NETWORK
TITLE = ---- Final
////////////////////////////////////////////////////////////////////////////////////////
////////////////////////////////////////////////////////////////////////////////////////
////////////////////////////////////////////////////////////////////////////////////////
// Se acabo el evento
Final_EventoRecibido_RefrescoUT:NOP   0;
      L     #P_Eventos;  // Recupero por donde voy en la lista de eventos
      LAR2;  // Regreso a buscar el siguiente evento
      JU    FinBucle_EventosRecibidos;



NETWORK
TITLE = Guardar Datos - Evento MOVE - Mover UT de Mesa // 08 02 2017
GuardarDatos_EventoRecibido_MOVE:NOP   0;

/////////////////////////////////////////////////////////////////////////
/////////////////////////////////////////////////////////////////////////
/////////////////////////////////////////////////////////////////////////
// --- Guardar Datos del Evento Recibido


/////////////////////////////////////////////////////////////////////////
/////////////////////////////////////////////////////////////////////////
/////////////////////////////////////////////////////////////////////////
// --- Control de Mesa Recibida
      L     #AtributosDeUTs.MesaActual;  // Ver que mesa es
      L     "CTE_OffsetMesa";
      -I;
      T     #VarTempUTs.MesaActual;

      L     #VarTempUTs.MesaActual;  // Comprobar el numero de mesa
      L     1;  // No menor de 1
      <I;  // No es correcto
      JC    Final_EventoRecibido_MOVE;
      L     #VarTempUTs.MesaActual;
      L     "CTE_MaxMesas";  // No mayor que el parametro
      >I;  // No es correcto
      JC    Final_EventoRecibido_MOVE;


///////////////////////////////////////////////////////////////////////////////
// --- Control de McKey Recibido
      L     #AtributosDeUTs.Mckey;  // Se ha recibido Mckey = 0
      L     0;  // No se puede Crear
      ==D;
      JC    Final_EventoRecibido_MOVE;


///////////////////////////////////////////////////////////////////////////////
// --- Busca el Mckey Recibido, comprobar que existe

      CALL  "FC720_BuscarUT_EnMesa"
      ( Mckey      := #AtributosDeUTs.Mckey,
        MesaActual := #VarTempUTs.MesaActual,
        NumeroUT   := #VarTempUTs.NumeroUT
      );

      L     #VarTempUTs.NumeroUT;
      L     0;
      ==I;  // No Existe UT ?
      JC    Final_EventoRecibido_MOVE;



NETWORK
TITLE = ---- Accion del Evento
///////////////////////////////////////////////////////////////////////////////
///////////////////////////////////////////////////////////////////////////////
///////////////////////////////////////////////////////////////////////////////
// --- Guardar Respuesta

      SET;
      L     "DB812_UTs_Control".UT[#VarTempUTs.NumeroUT].MesaActual;
      L     #AtributosDeUTs.MesaActual;
      <>I;  // Esta en Mesa diferente ?
      JC    Final_EventoRecibido_MOVE;

      SET;  // Realizada la peticion de Cambio de Mesa ?
      AN    "DB812_UTs_Control".UT[#VarTempUTs.NumeroUT].EventosDeCambioDeMesa.PeticionCambiarUTDeMesa;
      JC    Final_EventoRecibido_MOVE;


///////////////////////////////////////////////////////////////////////////////
///////////////////////////////////////////////////////////////////////////////
///////////////////////////////////////////////////////////////////////////////
// --- Orden Recibida guardarla en la UT

      SET;  // OK Cambiar UT de Mesa Final
      A     #AtributosDeUTs.CambiarUTDeMesa.OK;
      A     #AtributosDeUTs.CambiarUTDeMesa.Final;
      S     "DB812_UTs_Control".UT[#VarTempUTs.NumeroUT].EventosDeCambioDeMesa.OKCambiarUTDeMesaFinal;

      SET;  // OK Cambiar UT de Mesa Inicio
      A     #AtributosDeUTs.CambiarUTDeMesa.OK;
      A     #AtributosDeUTs.CambiarUTDeMesa.Inicio;
      S     "DB812_UTs_Control".UT[#VarTempUTs.NumeroUT].EventosDeCambioDeMesa.OKCambiarUTDeMesaInicio;

      SET;  // NOK Cambiar UT de Mesa
      A     #AtributosDeUTs.CambiarUTDeMesa.NOK;
      S     "DB812_UTs_Control".UT[#VarTempUTs.NumeroUT].EventosDeCambioDeMesa.NOKCambiarUTDeMesa;


///////////////////////////////////////////////////////////////////////////////
      JU    Final_EventoRecibido_MOVE;



NETWORK
TITLE = ---- Final
///////////////////////////////////////////////////////////////////////////////
///////////////////////////////////////////////////////////////////////////////
///////////////////////////////////////////////////////////////////////////////
// Se acabo el evento
Final_EventoRecibido_MOVE:NOP   0;
      L     #P_Eventos;  // Recupero por donde voy en la lista de eventos
      LAR2;
      JU    FinBucle_EventosRecibidos;



NETWORK
TITLE = Guardar Datos - Evento DEMB - Datos de EmBandejado de la UT // Fecha 07 06 2017
GuardarDatos_EventoRecibido_DEMB:NOP   0;

/////////////////////////////////////////////////////////////////////////
/////////////////////////////////////////////////////////////////////////
/////////////////////////////////////////////////////////////////////////
// --- Guardar Datos del Evento Recibido


/////////////////////////////////////////////////////////////////////////
/////////////////////////////////////////////////////////////////////////
/////////////////////////////////////////////////////////////////////////
// --- Control de Mesa Recibida
      L     #AtributosDeUTs.MesaActual;
      L     0;
      ==I;
      JC    FinControlMesa_EventoRecibido_DEMB;

      L     #AtributosDeUTs.MesaActual;  // Ver que mesa es
      L     "CTE_OffsetMesa";
      -I;
      T     #VarTempUTs.MesaActual;

      L     #VarTempUTs.MesaActual;  // Comprobar el numero de mesa
      L     1;  // No menor de 1
      <I;  // No es correcto
      JC    Final_EventoRecibido_DEMB;
      L     #VarTempUTs.MesaActual;
      L     "CTE_MaxMesas";  // No mayor que el parametro
      >I;  // No es correcto
      JC    Final_EventoRecibido_DEMB;

/////////////////////////////////////////////////////////////////////////
FinControlMesa_EventoRecibido_DEMB:NOP   0;


/////////////////////////////////////////////////////////////////////////
/////////////////////////////////////////////////////////////////////////
/////////////////////////////////////////////////////////////////////////
// --- Control de Mckey Recibido
      L     #AtributosDeUTs.Mckey;  // Se ha recibido Mckey = 0
      L     0;  // No se puede Crear
      ==D;
      JC    Final_EventoRecibido_DEMB;


/////////////////////////////////////////////////////////////////////////
/////////////////////////////////////////////////////////////////////////
/////////////////////////////////////////////////////////////////////////
// --- Comprobar que Existe una UT
      CALL  "FC720_BuscarUT_EnMesa"
      ( Mckey      := #AtributosDeUTs.Mckey,
        MesaActual := #VarTempUTs.MesaActual,
        NumeroUT   := #VarTempUTs.NumeroUT
      );

      L     #VarTempUTs.NumeroUT;
      L     0;
      ==I;  // No Existe UT ?
      JC    Final_EventoRecibido_DEMB;



NETWORK
TITLE = ---- Accion del Evento
/////////////////////////////////////////////////////////////////////////
/////////////////////////////////////////////////////////////////////////
/////////////////////////////////////////////////////////////////////////
// Guardar Respuesta


      L     #AtributosDeUTs.QUBIQA_NumeroBulto;  // Numero de Bulto
      T     "DB820_UTs_DatosQUBIQA".UT[#VarTempUTs.NumeroUT].NumeroDeBulto;
      L     #AtributosDeUTs.QUBIQA_TotalBultos;  // Numero de Bultos
      T     "DB820_UTs_DatosQUBIQA".UT[#VarTempUTs.NumeroUT].TotalBultos;

      CALL  BLKMOV
      ( SRCBLK  := #AtributosDeUTs.QUBIQA_PID,
        RET_VAL := #ReturnValor,
        DSTBLK  := "DB820_UTs_DatosQUBIQA".UT[#VarTempUTs.NumeroUT].PID
      );  // Guardar el PID

      JU    Final_EventoRecibido_DEMB;



NETWORK
TITLE = ---- Final
/////////////////////////////////////////////////////////////////////////
/////////////////////////////////////////////////////////////////////////
/////////////////////////////////////////////////////////////////////////
// Se acabo el evento
Final_EventoRecibido_DEMB:NOP   0;
      L     #P_Eventos;  // Recupero por donde voy en la lista de eventos
      LAR2;
      JU    FinBucle_EventosRecibidos;



NETWORK
TITLE = ////////////////////////////////////////////////////////////////////////////////////////////////////////////

NETWORK
TITLE = Evento CSTA - Notificacion de cambio de Estado de un dispositivo
// Analisis del evento
// - Inicializa variables de los atributos del Evento
// - Buscar Atributos o Final del Evento
// - Guardar datos del Evento
//   - Si es tipo CCPIF (50)
//   - Si es tipo CBOX (40)
//   - Si es tipo Mesa (60)
//   - Si es tipo Maquina (70)
// Analisis de los atributos de los eventos
// - Mirar que atributo del Evento es ?
// - Distribuir a recoger los datos del Evento
// - Recoger el Atributo Tipo de Dispositivo
// - Recoger el Atributo Numero de Dispositivo
// - Recoger el Atributo Nuevo Estado del Dispositivo
GuardarDatos_EventoRecibido_CSTA:NOP   0;

/////////////////////////////////////////////////////////////////////////
/////////////////////////////////////////////////////////////////////////
/////////////////////////////////////////////////////////////////////////
// --- Guardar Datos del Evento Recibido


/////////////////////////////////////////////////////////////////////////
/////////////////////////////////////////////////////////////////////////
/////////////////////////////////////////////////////////////////////////
// --- Repartir segun tipo de dispositivo: CCPIF, CBOX, Mesa ....

      SET;  // Es CCPIF
      L     #AtributosDeDispositivos.Tipo;
      L     50;
      ==I;
      JC    DispositivosCCPIF_EventoRecibido_CSTA;

      SET;  // Es CBOX
      L     #AtributosDeDispositivos.Tipo;
      L     40;
      ==I;
      JC    DispositivosCBOX_EventoRecibido_CSTA;

      SET;  // Es Mesa
      L     #AtributosDeDispositivos.Tipo;
      L     60;
      ==I;
      JC    DispositivosMesa_EventoRecibido_CSTA;

      SET;  // Es Baliza
      L     #AtributosDeDispositivos.Tipo;
      L     1000;
      ==I;
      JC    DispositivosBaliza_EventoRecibido_CSTA;

/////////////////////////////////////////////////////////////////////////
/////////////////////////////////////////////////////////////////////////
/////////////////////////////////////////////////////////////////////////

      SET;  // Es Llave
      L     #AtributosDeDispositivos.Tipo;
      L     1001;
      ==I;
      JC    DispositivosLlave_EventoRecibido_CSTA;

      SET;  // Es Seta
      L     #AtributosDeDispositivos.Tipo;
      L     1002;
      ==I;
      JC    DispositivosSeta_EventoRecibido_CSTA;

      SET;  // Es Barrera
      L     #AtributosDeDispositivos.Tipo;
      L     1003;
      ==I;
      JC    DispositivosBarrera_EventoRecibido_CSTA;

      SET;  // Es Puerta
      L     #AtributosDeDispositivos.Tipo;
      L     1004;
      ==I;
      JC    DispositivosPuerta_EventoRecibido_CSTA;

      SET;  // Es Linea de Potencia
      L     #AtributosDeDispositivos.Tipo;
      L     1005;
      ==I;
      JC    DispositivosLineaPotencia_EventoRecibido_CSTA;


/////////////////////////////////////////////////////////////////////////
/////////////////////////////////////////////////////////////////////////
/////////////////////////////////////////////////////////////////////////
// Es Maquina De 70 ... 99
      SET;
      A(;
      L     #AtributosDeDispositivos.Tipo;
      L     70;
      >=I;
      );
      A(;
      SET;
      L     #AtributosDeDispositivos.Tipo;
      L     99;
      <=I;
      );
      JC    DispositivosMaquina_EventoRecibido_CSTA;


/////////////////////////////////////////////////////////////////////////
/////////////////////////////////////////////////////////////////////////
/////////////////////////////////////////////////////////////////////////
// --- No es ningun Tipo de Dispositivo Esperado
      JU    Final_EventoRecibido_CSTA;



NETWORK
TITLE = ---- Accion del Evento --> Notificacion de cambio de Estado de CCPIF
///////////////////////////////////////////////////////////////////////////////
///////////////////////////////////////////////////////////////////////////////
///////////////////////////////////////////////////////////////////////////////
// --- Tipo CCPIF
DispositivosCCPIF_EventoRecibido_CSTA:NOP   0;


///////////////////////////////////////////////////////////////////////////////
// --- Comprobacion del Numero de Dispositivo
      L     #AtributosDeDispositivos.Numero;  // Comprobacion del numero de CCPIF
      L     "CTE_OffsetCCPIF";
      -I;
      L     1;
      <>I;  // Numero de CCPIF incorrecto
      JC    Final_EventoRecibido_CSTA;


///////////////////////////////////////////////////////////////////////////////
// --- Guardar el Cambio de Estado Recibido
      L     #AtributosDeDispositivos.NuevoEstado;  // EstadoDispo + 260 = Recibido Evento de Cambio de Estado
      L     260;  // Orden a guardar en el DB
      +I;
      T     "DB830_Dispositivos".Dispositivos[0].EstadoRecepcionEvento;


///////////////////////////////////////////////////////////////////////////////
// --- Finalizar
      JU    Final_EventoRecibido_CSTA;



NETWORK
TITLE = ---- Accion del Evento --> Notificacion de cambio de Estado de CBOX
///////////////////////////////////////////////////////////////////////////////
///////////////////////////////////////////////////////////////////////////////
///////////////////////////////////////////////////////////////////////////////
// --- Tipo CBOX
DispositivosCBOX_EventoRecibido_CSTA:NOP   0;


///////////////////////////////////////////////////////////////////////////////
// --- Comprobacion del Numero de Dispositivo
      L     #AtributosDeDispositivos.Numero;  // Comprobacion del numero de CCPIF
      L     100;
      /I;
      L     "CTE_OffsetCCPIF";
      -I;
      L     1;
      <>I;  // Numero de CCPIF incorrecto
      JC    Final_EventoRecibido_CSTA;


      L     #AtributosDeDispositivos.Numero;  // Calculo del numero de CBOX
      L     100;
      MOD;  // Var verlo en la DB_Dispositivos
      T     #VarTempDispositivos.Numero;

      L     #VarTempDispositivos.Numero;  // Comprobacion del numero de CBOX
      L     1;  // Es menor de 1
      <I;  // No es correcto el numero de CBOX
      JC    Final_EventoRecibido_CSTA;
      L     #VarTempDispositivos.Numero;
      L     "CTE_MaxDispositivos";  // Si es mayor que el parametro
      >I;  // No es correcto el numero de CBOX
      JC    Final_EventoRecibido_CSTA;


///////////////////////////////////////////////////////////////////////////////
// --- Guardar el Cambio de Estado Recibido
      L     #AtributosDeDispositivos.NuevoEstado;  // EstadoDispo + 260 = Recibido Evento de Cambio de Estado
      L     260;  // Orden a guardar en el DB
      +I;
      T     "DB830_Dispositivos".Dispositivos[#VarTempDispositivos.Numero].EstadoRecepcionEvento;


///////////////////////////////////////////////////////////////////////////////
// --- Finalizar
      JU    Final_EventoRecibido_CSTA;



NETWORK
TITLE = ---- Accion del Evento --> Notificacion de cambio de Estado de Mesa
///////////////////////////////////////////////////////////////////////////////
///////////////////////////////////////////////////////////////////////////////
///////////////////////////////////////////////////////////////////////////////
// --- Tipo Mesa
DispositivosMesa_EventoRecibido_CSTA:NOP   0;


///////////////////////////////////////////////////////////////////////////////
// --- Comprobacion del Numero de Dispositivo
      L     #AtributosDeDispositivos.Numero;  // Ver que mesa es
      L     "CTE_OffsetMesa";
      -I;
      T     #VarTempDispositivos.Numero;

      L     #VarTempDispositivos.Numero;  // Comprobar el numero de mesa
      L     1;  // No menor de 1
      <I;  // No es correcto
      JC    Final_EventoRecibido_CSTA;
      L     #VarTempDispositivos.Numero;
      L     "CTE_MaxMesas";  // No meyor que el parametro
      >I;  // No es correcto
      JC    Final_EventoRecibido_CSTA;


///////////////////////////////////////////////////////////////////////////////
// --- Guardar el Cambio de Estado Recibido
      L     #AtributosDeDispositivos.NuevoEstado;  // EstadoDispo + 260 = Recibido Evento de Cambio de Estado
      L     260;  // Orden a guardar en el DB
      +I;
      T     "DB831_Mesas".Mesas[#VarTempDispositivos.Numero].EstadoRecepcionEvento;


///////////////////////////////////////////////////////////////////////////////
// --- Habilitado o DesHabilitado el Dispositivo
      SET;
      L     #AtributosDeDispositivos.Habilitado;
      L     2001;  // Habitar Disposito = 0
      ==I;
      R     "DB831_Mesas".Mesas[#VarTempDispositivos.Numero].Memorias.DesHabilitado;

      SET;
      L     #AtributosDeDispositivos.Habilitado;
      L     2002;  // DesHabitar Disposito = 1
      ==I;
      S     "DB831_Mesas".Mesas[#VarTempDispositivos.Numero].Memorias.DesHabilitado;


///////////////////////////////////////////////////////////////////////////////
// Prioridad  - 1...x
      SET;
      L     #AtributosDeDispositivos.Prioridad;
      L     0;
      ==I;
      JC    SinPrioridadMesa_EventoRecibido_CSTA;

      L     #AtributosDeDispositivos.Prioridad;
      T     "DB831_Mesas".Mesas[#VarTempDispositivos.Numero].Prioridad;

SinPrioridadMesa_EventoRecibido_CSTA:NOP   0;


///////////////////////////////////////////////////////////////////////////////
// --- Fecha: 08 02 2017
// --- Motivo para la pantalla del Error envio por el JDT
      SET;
      L     #LonguitudTextoRecibido;
      L     0;
      ==I;  // Existe Motivo de Error en Mesa Enviado por el JDT
      JC    SinMotivoDeErrorDelJdT_EventoRecibido_CSTA;

      CALL  BLKMOV
      ( SRCBLK  := #AtributosDeDispositivos.MotivoDelError,
        RET_VAL := #ReturnValor,
        DSTBLK  := "DB907_TextoErrorJdT".Mesa[#VarTempDispositivos.Numero]
      );

SinMotivoDeErrorDelJdT_EventoRecibido_CSTA:NOP   0;


///////////////////////////////////////////////////////////////////////////////
// --- Finalizar
      JU    Final_EventoRecibido_CSTA;



NETWORK
TITLE = ---- Accion del Evento --> Notificacion de cambio de Estado de Maquina
///////////////////////////////////////////////////////////////////////////////
///////////////////////////////////////////////////////////////////////////////
///////////////////////////////////////////////////////////////////////////////
// --- Tipo Maquina
DispositivosMaquina_EventoRecibido_CSTA:NOP   0;


///////////////////////////////////////////////////////////////////////////////
// --- Comprobacion del Numero de Dispositivo
      L     #AtributosDeDispositivos.Numero;  // Ver que mesa es
      L     "CTE_OffsetMesa";
      -I;
      T     #VarTempDispositivos.Numero;

      L     #VarTempDispositivos.Numero;  // Comprobar el numero de maquina
      L     1;  // No menor de 1
      <I;  // No es correcto
      JC    Final_EventoRecibido_CSTA;
      L     #VarTempDispositivos.Numero;
      L     "CTE_MaxMesas";  // No meyor que el parametro
      >I;  // No es correcto
      JC    Final_EventoRecibido_CSTA;


///////////////////////////////////////////////////////////////////////////////
// --- Guardar el Cambio de Estado Recibido

      L     #AtributosDeDispositivos.NuevoEstado;  // EstadoDispo + 260 = Recibido Evento de Cambio de Estado
      L     260;  // Orden a guardar en el DB
      +I;
      T     "DB832_Maquinas".Maquinas[#VarTempDispositivos.Numero].EstadoRecepcionEvento;


///////////////////////////////////////////////////////////////////////////////
// --- Habilitado o DesHabilitado
      SET;
      L     #AtributosDeDispositivos.Habilitado;
      L     2001;  // Habitar Disposito = 0
      ==I;
      R     "DB832_Maquinas".Maquinas[#VarTempDispositivos.Numero].Memorias.DesHabilitado;

      SET;
      L     #AtributosDeDispositivos.Habilitado;
      L     2002;  // DesHabitar Disposito = 1
      ==I;
      S     "DB832_Maquinas".Maquinas[#VarTempDispositivos.Numero].Memorias.DesHabilitado;


///////////////////////////////////////////////////////////////////////////////
// Prioridad  - 1...x
      SET;
      L     #AtributosDeDispositivos.Prioridad;
      L     0;
      ==I;
      JC    SinPrioridadMaquina_EventoRecibido_CSTA;

      L     #AtributosDeDispositivos.Prioridad;
      T     "DB832_Maquinas".Maquinas[#VarTempDispositivos.Numero].Prioridad;

SinPrioridadMaquina_EventoRecibido_CSTA:NOP   0;


///////////////////////////////////////////////////////////////////////////////
// Finalizar
      JU    Final_EventoRecibido_CSTA;



NETWORK
TITLE = ---- Accion del Evento --> Notificacion de cambio de Estado de Baliza
///////////////////////////////////////////////////////////////////////////////
///////////////////////////////////////////////////////////////////////////////
///////////////////////////////////////////////////////////////////////////////
// --- Tipo Baliza
DispositivosBaliza_EventoRecibido_CSTA:NOP   0;


///////////////////////////////////////////////////////////////////////////////
// --- Comprobacion del Numero de Dispositivo
      L     #AtributosDeDispositivos.Numero;  // Ver que Baliza es
      L     "CTE_OffsetMesa";
      -I;
      T     #VarTempDispositivos.Numero;

      L     #VarTempDispositivos.Numero;  // Comprobar el numero de Baliza
      L     1;  // No menor de 1
      <I;  // No es correcto
      JC    Final_EventoRecibido_CSTA;
      L     #VarTempDispositivos.Numero;
      L     "CTE_MaxDispositivosBaliza";  // No meyor que el parametro
      >I;  // No es correcto
      JC    Final_EventoRecibido_CSTA;


///////////////////////////////////////////////////////////////////////////////
// --- Guardar el Cambio de Estado Recibido

      CALL  BLKMOV
      ( SRCBLK  := "DB839_DispositivosVarios".DispoBaliza[#VarTempDispositivos.Numero],
        RET_VAL := #ReturnValor,
        DSTBLK  := #VarTempDispositivos.Baliza
      );

      SET;  // Reseteo para actualizar
      R     #VarTempDispositivos.Baliza.Sonoro;
      R     #VarTempDispositivos.Baliza.Verde;
      R     #VarTempDispositivos.Baliza.Rojo;
      R     #VarTempDispositivos.Baliza.Amarillo;
      R     #VarTempDispositivos.Baliza.Azul;


      SET;  // Sonoro
      A     #AtributosDeDispositivos.BalizaColor.Sonoro;
      S     #VarTempDispositivos.Baliza.Sonoro;

      SET;  // Verde
      A     #AtributosDeDispositivos.BalizaColor.Verde;
      S     #VarTempDispositivos.Baliza.Verde;

      SET;  // Rojo
      A     #AtributosDeDispositivos.BalizaColor.Rojo;
      S     #VarTempDispositivos.Baliza.Rojo;

      SET;  // Amarillo
      A     #AtributosDeDispositivos.BalizaColor.Amarillo;
      S     #VarTempDispositivos.Baliza.Amarillo;

      SET;  // Azul
      A     #AtributosDeDispositivos.BalizaColor.Azul;
      S     #VarTempDispositivos.Baliza.Azul;

      SET;  // Peticion de Estado
      S     #VarTempDispositivos.Baliza.RefrescoDatos;

      CALL  BLKMOV
      ( SRCBLK  := #VarTempDispositivos.Baliza,
        RET_VAL := #ReturnValor,
        DSTBLK  := "DB839_DispositivosVarios".DispoBaliza[#VarTempDispositivos.Numero]
      );


///////////////////////////////////////////////////////////////////////////////
// Finalizar
      JU    Final_EventoRecibido_CSTA;



NETWORK
TITLE = ---- Accion del Evento --> Notificacion de cambio de Estado de Llave
///////////////////////////////////////////////////////////////////////////////
///////////////////////////////////////////////////////////////////////////////
///////////////////////////////////////////////////////////////////////////////
// --- Tipo Llave
DispositivosLlave_EventoRecibido_CSTA:NOP   0;


///////////////////////////////////////////////////////////////////////////////
// --- Comprobacion del Numero de Dispositivo
      L     #AtributosDeDispositivos.Numero;  // Ver que Llave es
      L     "CTE_OffsetMesa";
      -I;
      T     #VarTempDispositivos.Numero;

      L     #VarTempDispositivos.Numero;  // Comprobar el numero de Llave
      L     1;  // No menor de 1
      <I;  // No es correcto
      JC    Final_EventoRecibido_CSTA;
      L     #VarTempDispositivos.Numero;
      L     "CTE_MaxDispositivosLlave";  // No meyor que el parametro
      >I;  // No es correcto
      JC    Final_EventoRecibido_CSTA;


///////////////////////////////////////////////////////////////////////////////
// --- Guardar el Cambio de Estado Recibido

      SET;
      S     "DB839_DispositivosVarios".DispoLlave[#VarTempDispositivos.Numero].Habilitado;  // Por defecto DesHabilitado

      L     #AtributosDeDispositivos.Habilitado;
      L     2001;  // Nuevo estado - Habilitado SI ?
      ==I;
      JC    HabilitadaLlave_EventoRecibido_CSTA;

      SET;
      R     "DB839_DispositivosVarios".DispoLlave[#VarTempDispositivos.Numero].Habilitado;

HabilitadaLlave_EventoRecibido_CSTA:NOP   0;

      SET;
      S     "DB839_DispositivosVarios".DispoLlave[#VarTempDispositivos.Numero].RefrescoDatos;  // Peticion de Refresco de datos


///////////////////////////////////////////////////////////////////////////////
// Finalizar
      JU    Final_EventoRecibido_CSTA;



NETWORK
TITLE = ---- Accion del Evento --> Notificacion de cambio de Estado de Seta
///////////////////////////////////////////////////////////////////////////////
///////////////////////////////////////////////////////////////////////////////
///////////////////////////////////////////////////////////////////////////////
// --- Tipo Seta
DispositivosSeta_EventoRecibido_CSTA:NOP   0;


///////////////////////////////////////////////////////////////////////////////
// --- Comprobacion del Numero de Dispositivo
      L     #AtributosDeDispositivos.Numero;  // Ver que Seta es
      L     "CTE_OffsetMesa";
      -I;
      T     #VarTempDispositivos.Numero;

      L     #VarTempDispositivos.Numero;  // Comprobar el numero de Seta
      L     1;  // No menor de 1
      <I;  // No es correcto
      JC    Final_EventoRecibido_CSTA;
      L     #VarTempDispositivos.Numero;
      L     "CTE_MaxDispositivosSeta";  // No meyor que el parametro
      >I;  // No es correcto
      JC    Final_EventoRecibido_CSTA;


///////////////////////////////////////////////////////////////////////////////
// --- Guardar el Cambio de Estado Recibido

      SET;
      S     "DB839_DispositivosVarios".DispoSeta[#VarTempDispositivos.Numero].Habilitado;  // Por defecto DesHabilitado

      L     #AtributosDeDispositivos.Habilitado;
      L     2001;  // Nuevo estado - Habilitado SI ?
      ==I;
      JC    HabilitadaSeta_EventoRecibido_CSTA;

      SET;
      R     "DB839_DispositivosVarios".DispoSeta[#VarTempDispositivos.Numero].Habilitado;

HabilitadaSeta_EventoRecibido_CSTA:NOP   0;

      SET;
      S     "DB839_DispositivosVarios".DispoSeta[#VarTempDispositivos.Numero].RefrescoDatos;  // Peticion de Refresco de datos


///////////////////////////////////////////////////////////////////////////////
// Finalizar
      JU    Final_EventoRecibido_CSTA;



NETWORK
TITLE = ---- Accion del Evento --> Notificacion de cambio de Estado de Barrera
///////////////////////////////////////////////////////////////////////////////
///////////////////////////////////////////////////////////////////////////////
///////////////////////////////////////////////////////////////////////////////
// --- Tipo Barrera
DispositivosBarrera_EventoRecibido_CSTA:NOP   0;


///////////////////////////////////////////////////////////////////////////////
// --- Comprobacion del Numero de Dispositivo
      L     #AtributosDeDispositivos.Numero;  // Ver que Barrera es
      L     "CTE_OffsetMesa";
      -I;
      T     #VarTempDispositivos.Numero;

      L     #VarTempDispositivos.Numero;  // Comprobar el numero de Barrera
      L     1;  // No menor de 1
      <I;  // No es correcto
      JC    Final_EventoRecibido_CSTA;
      L     #VarTempDispositivos.Numero;
      L     "CTE_MaxDispositivosBarrera";  // No meyor que el parametro
      >I;  // No es correcto
      JC    Final_EventoRecibido_CSTA;


///////////////////////////////////////////////////////////////////////////////
// --- Guardar el Cambio de Estado Recibido

      SET;
      S     "DB839_DispositivosVarios".DispoBarrera[#VarTempDispositivos.Numero].Habilitado;  // Por defecto DesHabilitado

      L     #AtributosDeDispositivos.Habilitado;
      L     2001;  // Nuevo estado - Habilitado SI ?
      ==I;
      JC    HabilitadaBarrera_EventoRecibido_CSTA;

      SET;
      R     "DB839_DispositivosVarios".DispoBarrera[#VarTempDispositivos.Numero].Habilitado;

HabilitadaBarrera_EventoRecibido_CSTA:NOP   0;

      SET;
      S     "DB839_DispositivosVarios".DispoBarrera[#VarTempDispositivos.Numero].RefrescoDatos;  // Peticion de Refresco de datos


///////////////////////////////////////////////////////////////////////////////
// Finalizar
      JU    Final_EventoRecibido_CSTA;



NETWORK
TITLE = ---- Accion del Evento --> Notificacion de cambio de Estado de Puerta
///////////////////////////////////////////////////////////////////////////////
///////////////////////////////////////////////////////////////////////////////
///////////////////////////////////////////////////////////////////////////////
// --- Tipo Puerta
DispositivosPuerta_EventoRecibido_CSTA:NOP   0;


///////////////////////////////////////////////////////////////////////////////
// --- Comprobacion del Numero de Dispositivo
      L     #AtributosDeDispositivos.Numero;  // Ver que Puerta es
      L     "CTE_OffsetMesa";
      -I;
      T     #VarTempDispositivos.Numero;

      L     #VarTempDispositivos.Numero;  // Comprobar el numero de Puerta
      L     1;  // No menor de 1
      <I;  // No es correcto
      JC    Final_EventoRecibido_CSTA;
      L     #VarTempDispositivos.Numero;
      L     "CTE_MaxDispositivosPuerta";  // No meyor que el parametro
      >I;  // No es correcto
      JC    Final_EventoRecibido_CSTA;


///////////////////////////////////////////////////////////////////////////////
// --- Guardar el Cambio de Estado Recibido

      SET;
      S     "DB839_DispositivosVarios".DispoPuerta[#VarTempDispositivos.Numero].Habilitado;  // Por defecto DesHabilitado

      L     #AtributosDeDispositivos.Habilitado;
      L     2001;  // Nuevo estado - Habilitado SI ?
      ==I;
      JC    HabilitadaPuerta_EventoRecibido_CSTA;

      SET;
      R     "DB839_DispositivosVarios".DispoPuerta[#VarTempDispositivos.Numero].Habilitado;

HabilitadaPuerta_EventoRecibido_CSTA:NOP   0;

      SET;
      S     "DB839_DispositivosVarios".DispoPuerta[#VarTempDispositivos.Numero].RefrescoDatos;  // Peticion de Refresco de datos


///////////////////////////////////////////////////////////////////////////////
// Finalizar
      JU    Final_EventoRecibido_CSTA;



NETWORK
TITLE = ---- Accion del Evento --> Notificacion de cambio de Estado de Linea de Potencia
///////////////////////////////////////////////////////////////////////////////
///////////////////////////////////////////////////////////////////////////////
///////////////////////////////////////////////////////////////////////////////
// --- Tipo Linea de Potencia
DispositivosLineaPotencia_EventoRecibido_CSTA:NOP   0;


///////////////////////////////////////////////////////////////////////////////
// --- Comprobacion del Numero de Dispositivo
      L     #AtributosDeDispositivos.Numero;  // Ver que Linea de Potencia es
      L     "CTE_OffsetMesa";
      -I;
      T     #VarTempDispositivos.Numero;

      L     #VarTempDispositivos.Numero;  // Comprobar el numero de Linea de Potencia
      L     1;  // No menor de 1
      <I;  // No es correcto
      JC    Final_EventoRecibido_CSTA;
      L     #VarTempDispositivos.Numero;
      L     "CTE_MaxDispositivosLlave";  // No meyor que el parametro
      >I;  // No es correcto
      JC    Final_EventoRecibido_CSTA;


///////////////////////////////////////////////////////////////////////////////
// --- Guardar el Cambio de Estado Recibido

      SET;
      S     "DB839_DispositivosVarios".DispoLineaPotencia[#VarTempDispositivos.Numero].Habilitado;  // Por defecto DesHabilitado

      L     #AtributosDeDispositivos.Habilitado;
      L     2001;  // Nuevo estado - Habilitado SI ?
      ==I;
      JC    HabilitadaLineaPotencia_EventoRecibido_CSTA;

      SET;
      R     "DB839_DispositivosVarios".DispoLineaPotencia[#VarTempDispositivos.Numero].Habilitado;

HabilitadaLineaPotencia_EventoRecibido_CSTA:NOP   0;

      SET;
      S     "DB839_DispositivosVarios".DispoLineaPotencia[#VarTempDispositivos.Numero].RefrescoDatos;  // Peticion de Refresco de datos


///////////////////////////////////////////////////////////////////////////////
// Finalizar
      JU    Final_EventoRecibido_CSTA;



NETWORK
TITLE = ---- Final
///////////////////////////////////////////////////////////////////////////////
///////////////////////////////////////////////////////////////////////////////
///////////////////////////////////////////////////////////////////////////////
// Se acabo el evento
Final_EventoRecibido_CSTA:NOP   0;
      L     #P_Eventos;  // Recupero por donde voy en la lista de eventos
      LAR2;
      JU    FinBucle_EventosRecibidos;  // Regreso a buscar el siguiente evento



NETWORK
TITLE = Evento ¿ST? - Peticion de Refresco de los dispositivos
// - Inicializa variables de los atributos del Evento
// - Buscar Atributos o Final del Evento
// - Guardar datos del Evento
//   - Si tiene Tipo y Numero
//   - Si solo Tipo
//   - Si son todos
GuardarDatos_EventoRecibido_Refresco_ST:NOP   0;

/////////////////////////////////////////////////////////////////////////
/////////////////////////////////////////////////////////////////////////
/////////////////////////////////////////////////////////////////////////
// --- Guardar Datos del Evento Recibido
/////////////////////////////////////////////////////////////////////////
/////////////////////////////////////////////////////////////////////////
/////////////////////////////////////////////////////////////////////////
// --- Distribucion por tipo

      SET;  // Dispositivo CCPIF
      L     #AtributosDeDispositivos.Tipo;
      L     50;
      ==I;
      JC    DispositivoCCPIF_EventoRecibido_RefrescoDispositivo;

      SET;  // Dispositivo CBOX
      L     #AtributosDeDispositivos.Tipo;
      L     40;
      ==I;
      JC    DispositivoCBOX_EventoRecibido_RefrescoDispositivo;

      SET;  // Dispositivo Mesa
      L     #AtributosDeDispositivos.Tipo;
      L     60;
      ==I;
      JC    DispositivoMesa_EventoRecibido_RefrescoDispositivo;


///////////////////////////////////////////////////////////////////////////////
///////////////////////////////////////////////////////////////////////////////
///////////////////////////////////////////////////////////////////////////////

      SET;  // Dispositivos Baliza
      L     #AtributosDeDispositivos.Tipo;
      L     1000;
      ==I;
      JC    DispositivoBaliza_EventoRecibido_RefrescoDispositivo;

      SET;  // Dispositivos Llave
      L     #AtributosDeDispositivos.Tipo;
      L     1001;
      ==I;
      JC    DispositivoLlave_EventoRecibido_RefrescoDispositivo;

      SET;  // Dispositivos Seta
      L     #AtributosDeDispositivos.Tipo;
      L     1002;
      ==I;
      JC    DispositivoSeta_EventoRecibido_RefrescoDispositivo;

      SET;  // Dispositivos Barrera
      L     #AtributosDeDispositivos.Tipo;
      L     1003;
      ==I;
      JC    DispositivoBarrera_EventoRecibido_RefrescoDispositivo;

      SET;  // Dispositivos Puerta
      L     #AtributosDeDispositivos.Tipo;
      L     1004;
      ==I;
      JC    DispositivoPuerta_EventoRecibido_RefrescoDispositivo;

      SET;  // Dispositivos Linea de Potencia
      L     #AtributosDeDispositivos.Tipo;
      L     1005;
      ==I;
      JC    DispositivoLineaPotencia_EventoRecibido_RefrescoDispositivo;


///////////////////////////////////////////////////////////////////////////////
///////////////////////////////////////////////////////////////////////////////
///////////////////////////////////////////////////////////////////////////////
// Dispositivo Maquina De 70 ... 99
      SET;
      A(;
      L     #AtributosDeDispositivos.Tipo;
      L     70;
      >=I;
      );
      A(;
      L     #AtributosDeDispositivos.Tipo;
      L     99;
      <=I;
      );
      JC    DispositivoMaquina_EventoRecibido_RefrescoDispositivo;


///////////////////////////////////////////////////////////////////////////////
///////////////////////////////////////////////////////////////////////////////
///////////////////////////////////////////////////////////////////////////////
// --- Todos los dipositivos -> Por defecto
      JU    DispositivosTodos_EventoRecibido_RefrescoDispositivo;



NETWORK
TITLE = ---- Accion del Evento --> Peticion de Refresco del Dispositivo CCPIF
///////////////////////////////////////////////////////////////////////////////
///////////////////////////////////////////////////////////////////////////////
///////////////////////////////////////////////////////////////////////////////
// Dispositivos tipo CCPIF
DispositivoCCPIF_EventoRecibido_RefrescoDispositivo:NOP   0;
      SET;
      L     #AtributosDeDispositivos.Numero;  // No se envia Numero CCPIF
      L     0;  // Son todos los CCPIF's (Solo uno)
      ==I;
      JC    RefrescoDipositivoCCPIF_RefrescoDispositivo_EventosRecibidos;

      L     #AtributosDeDispositivos.Numero;  // Comprobacion del numero de CCPIF
      L     "CTE_OffsetCCPIF";
      -I;
      L     1;
      <>I;  // Numero de CCPIF incorrecto
      JC    Final_EventoRecibido_RefrescoDispositivo;


///////////////////////////////////////////////////////////////////////////////
// Activar Refresco del Dispositivo
RefrescoDipositivoCCPIF_RefrescoDispositivo_EventosRecibidos:NOP   0;

      L     250;  // 250 - Recibido Evento de Refresco de Datos del Dispositivo
      T     "DB830_Dispositivos".Dispositivos[0].EstadoRecepcionEvento;


///////////////////////////////////////////////////////////////////////////////
// Finalizar
      JU    Final_EventoRecibido_RefrescoDispositivo;



NETWORK
TITLE = ---- Accion del Evento --> Peticion de Refresco del Dispositivo CBOX
///////////////////////////////////////////////////////////////////////////////
///////////////////////////////////////////////////////////////////////////////
///////////////////////////////////////////////////////////////////////////////
// --- Dispositivos tipo CBOX, uno determinado o todos
DispositivoCBOX_EventoRecibido_RefrescoDispositivo:NOP   0;
      SET;
      L     #AtributosDeDispositivos.Numero;  // Mirar si hay numero de CBOX
      L     0;  // Son todos los CBOX's
      ==I;
      JC    DispositivosTodosCBOX_EventoRecibido_RefrescoDispositivo;


///////////////////////////////////////////////////////////////////////////////
// --- Es Un CBOX Determinado
      JU    DispositivoUnCBOX_EventoRecibido_RefrescoDispositivo;



NETWORK
TITLE = ---- ---- De un CBOX
///////////////////////////////////////////////////////////////////////////////
///////////////////////////////////////////////////////////////////////////////
///////////////////////////////////////////////////////////////////////////////
// --- Un CBOX determinado
DispositivoUnCBOX_EventoRecibido_RefrescoDispositivo:NOP   0;


///////////////////////////////////////////////////////////////////////////////
// --- Comprobacion del numero de CCPIF
      L     #AtributosDeDispositivos.Numero;
      L     100;
      /I;
      L     "CTE_OffsetCCPIF";
      -I;
      L     1;
      <>I;  // Numero de CCPIF incorrecto
      JC    Final_EventoRecibido_RefrescoDispositivo;

      L     #AtributosDeDispositivos.Numero;  // Calculo del numero de CBOX
      L     100;
      MOD;  // Var verlo en la DB_Dispositivos
      T     #VarTempDispositivos.Numero;

      L     #VarTempDispositivos.Numero;  // Comprobacion del numero de CBOX
      L     1;  // Es menor de 1
      <I;  // No es correcto el numero de CBOX
      JC    Final_EventoRecibido_RefrescoDispositivo;
      L     #VarTempDispositivos.Numero;
      L     "CTE_MaxDispositivos";  // Si es mayor que el parametro
      >I;  // No es correcto el nuemro de CBOX
      JC    Final_EventoRecibido_RefrescoDispositivo;


///////////////////////////////////////////////////////////////////////////////
// --- Activar Refresco del Dispositivo
      L     250;  // 250 - Recibido Evento de Refresco de Datos del Dispositivo
      T     "DB830_Dispositivos".Dispositivos[#VarTempDispositivos.Numero].EstadoRecepcionEvento;


///////////////////////////////////////////////////////////////////////////////
// --- Finalizar
      JU    Final_EventoRecibido_RefrescoDispositivo;



NETWORK
TITLE = ---- ---- De Todos los CBOX
///////////////////////////////////////////////////////////////////////////////
///////////////////////////////////////////////////////////////////////////////
///////////////////////////////////////////////////////////////////////////////
// --- Son todos los CBOX
DispositivosTodosCBOX_EventoRecibido_RefrescoDispositivo:NOP   0;
      L     1;
      T     #IndiceCBOX;


///////////////////////////////////////////////////////////////////////////////
///////////////////////////////////////////////////////////////////////////////
///////////////////////////////////////////////////////////////////////////////
// --- Recorrer todo los dispositivos
BucleDispositivosTodosCBOX_EventoRecibido_RefrescoDispositivo:NOP   0;

// Mirar si Pertenece al JDT
      SET;
      X     "DB855_DefinicionDispositivos".Dispositivos[#IndiceCBOX].EventosDelJdT02;
      XN    #JDT02_Activo;
      =     #DispositivoDeJDT02;

      SET;
      AN    #DispositivoDeJDT02;
      JC    ContinuarBucleDispositivosTodosCBOX_EventoRecibido_RefrescoDispositivo;


///////////////////////////////////////////////////////////////////////////////
// Activar Refresco del Dispositivo
      L     250;  // 250 - Recibido Evento de Refresco de Datos del Dispositivo
      T     "DB830_Dispositivos".Dispositivos[#IndiceCBOX].EstadoRecepcionEvento;


///////////////////////////////////////////////////////////////////////////////
// Ir hacia el siguiente CBOX
ContinuarBucleDispositivosTodosCBOX_EventoRecibido_RefrescoDispositivo:NOP   0;
      L     #IndiceCBOX;  // Incremento al siguiente CBOX
      L     1;
      +I;
      T     #IndiceCBOX;

      L     #IndiceCBOX;
      L     "CTE_MaxDispositivos";
      >I;  // Finalizar
      JC    Final_EventoRecibido_RefrescoDispositivo;

///////////////////////////////////////////////////////////////////////////////
      JU    BucleDispositivosTodosCBOX_EventoRecibido_RefrescoDispositivo;



NETWORK
TITLE = ---- Accion del Evento --> Peticion de Refresco del Dispositivo Mesa
///////////////////////////////////////////////////////////////////////////////
///////////////////////////////////////////////////////////////////////////////
///////////////////////////////////////////////////////////////////////////////
// --- Dispositivos tipo Mesa, uno determinado o todos
DispositivoMesa_EventoRecibido_RefrescoDispositivo:NOP   0;
      SET;
      L     #AtributosDeDispositivos.Numero;  // Mirar si hay numero de Mesas
      L     0;  // Son todos los Mesas
      ==I;
      JC    DispositivosTodosMesa_EventoRecibido_RefrescoDispositivo;


///////////////////////////////////////////////////////////////////////////////
// --- Es Una Mesa Determinada
      JU    DispositivosUnaMesa_EventoRecibido_RefrescoDispositivo;




NETWORK
TITLE = ---- ---- De una Mesa
///////////////////////////////////////////////////////////////////////////////
///////////////////////////////////////////////////////////////////////////////
///////////////////////////////////////////////////////////////////////////////
// --- Una Mesa determinada
DispositivosUnaMesa_EventoRecibido_RefrescoDispositivo:NOP   0;

      L     #AtributosDeDispositivos.Numero;  // Ver que mesa es
      L     "CTE_OffsetMesa";
      -I;
      T     #VarTempDispositivos.Numero;

      L     #VarTempDispositivos.Numero;  // Comprobar el numero de mesa
      L     1;  // No menor de 1
      <I;  // No es correcto
      JC    Final_EventoRecibido_RefrescoDispositivo;
      L     #VarTempDispositivos.Numero;
      L     "CTE_MaxMesas";  // No meyor que el parametro
      >I;  // No es correcto
      JC    Final_EventoRecibido_RefrescoDispositivo;


///////////////////////////////////////////////////////////////////////////////
// --- Activar Refresco del Dispositivo
      L     250;  // 250 - Recibido Evento de Refresco de Datos del Dispositivo
      T     "DB831_Mesas".Mesas[#VarTempDispositivos.Numero].EstadoRecepcionEvento;


///////////////////////////////////////////////////////////////////////////////
// --- Finalizar
      JU    Final_EventoRecibido_RefrescoDispositivo;



NETWORK
TITLE = ---- ---- De Todas las Mesas
///////////////////////////////////////////////////////////////////////////////
///////////////////////////////////////////////////////////////////////////////
///////////////////////////////////////////////////////////////////////////////
// --- Todas las Mesas
DispositivosTodosMesa_EventoRecibido_RefrescoDispositivo:NOP   0;
      L     1;
      T     #IndiceMesa;


///////////////////////////////////////////////////////////////////////////////
///////////////////////////////////////////////////////////////////////////////
///////////////////////////////////////////////////////////////////////////////
// Recorrer todo los dispositivos
BucleDispositivosTodosMesa_EventoRecibido_RefrescoDispositivo:NOP   0;


///////////////////////////////////////////////////////////////////////////////
// Mirar si esta definido como mesa de Tracking y TL
      SET;
      AN    "DB850_DefinicionMesas".Mesa[#IndiceMesa].ConfigMesa.MesaPaso;
      AN    "DB850_DefinicionMesas".Mesa[#IndiceMesa].ConfigMesa.MesaCruce;
      AN    "DB850_DefinicionMesas".Mesa[#IndiceMesa].ConfigMesa.MesaMultiplesDestinos;
      AN    "DB850_DefinicionMesas".Mesa[#IndiceMesa].ConfigMesa.MesaTL;
      JC    ContinuarBucleDispositivosTodosMesa_EventoRecibido_RefrescoDispositivo;


///////////////////////////////////////////////////////////////////////////////
/// Mirar Si pertenece al JDT
      SET;
      X     "DB850_DefinicionMesas".Mesa[#IndiceMesa].ConfigMesa.MesaDeJDT02;  // JDT01 ?
      XN    #JDT02_Activo;
      =     #DispositivoDeJDT02;

      SET;
      AN    #DispositivoDeJDT02;
      JC    ContinuarBucleDispositivosTodosMesa_EventoRecibido_RefrescoDispositivo;


///////////////////////////////////////////////////////////////////////////////
// Activar Refresco del Dispositivo
      L     250;  // 250 - Recibido Evento de Refresco de Datos del Dispositivo
      T     "DB831_Mesas".Mesas[#IndiceMesa].EstadoRecepcionEvento;


///////////////////////////////////////////////////////////////////////////////
ContinuarBucleDispositivosTodosMesa_EventoRecibido_RefrescoDispositivo:NOP   0;
      L     #IndiceMesa;  // Incremento al siguiente Mesa
      L     1;
      +I;
      T     #IndiceMesa;

      L     #IndiceMesa;
      L     "CTE_MaxMesas";
      >I;  // Finalizar
      JC    Final_EventoRecibido_RefrescoDispositivo;


///////////////////////////////////////////////////////////////////////////////
// -- Ir hacia el siguiente Mesa
      JU    BucleDispositivosTodosMesa_EventoRecibido_RefrescoDispositivo;



NETWORK
TITLE = ---- Accion del Evento --> Peticion de Refresco del Dispositivo Maquinas
///////////////////////////////////////////////////////////////////////////////
///////////////////////////////////////////////////////////////////////////////
///////////////////////////////////////////////////////////////////////////////
// Dispositivos tipo Maquina uno determinado o todos
DispositivoMaquina_EventoRecibido_RefrescoDispositivo:NOP   0;
      SET;
      L     #AtributosDeDispositivos.Numero;  // Mirar si hay numero de maquina
      L     0;  // Son todos los CBOX's
      ==I;
      JC    DispositivosTodosMaquina_EventoRecibido_RefrescoDispositivo;


///////////////////////////////////////////////////////////////////////////////
// --- Es Una Maquina Determinada
      JU    DispositivosUnaMaquina_EventoRecibido_RefrescoDispositivo;



NETWORK
TITLE = ---- ---- De una Maquina
///////////////////////////////////////////////////////////////////////////////
///////////////////////////////////////////////////////////////////////////////
///////////////////////////////////////////////////////////////////////////////
// --- Maquina  determinada
DispositivosUnaMaquina_EventoRecibido_RefrescoDispositivo:NOP   0;

      L     #AtributosDeDispositivos.Numero;  // Ver que maquina es
      L     "CTE_OffsetMesa";
      -I;
      T     #VarTempDispositivos.Numero;

      L     #VarTempDispositivos.Numero;  // Comprobar el numero de maquina
      L     1;  // No menor de 1
      <I;  // No es correcto
      JC    Final_EventoRecibido_RefrescoDispositivo;
      L     #VarTempDispositivos.Numero;
      L     "CTE_MaxMesas";  // No meyor que el parametro
      >I;  // No es correcto
      JC    Final_EventoRecibido_RefrescoDispositivo;


///////////////////////////////////////////////////////////////////////////////
// --- Activar Refresco del Dispositivo
      L     250;  // 250 - Recibido Evento de Refresco de Datos del Dispositivo
      T     "DB832_Maquinas".Maquinas[#VarTempDispositivos.Numero].EstadoRecepcionEvento;


///////////////////////////////////////////////////////////////////////////////
// --- Finalizar
      JU    Final_EventoRecibido_RefrescoDispositivo;



NETWORK
TITLE = ---- ---- De Todas las Maquinas
///////////////////////////////////////////////////////////////////////////////
///////////////////////////////////////////////////////////////////////////////
///////////////////////////////////////////////////////////////////////////////
// --- Todas las Maquinas
DispositivosTodosMaquina_EventoRecibido_RefrescoDispositivo:NOP   0;
      L     1;
      T     #IndiceMaquina;


///////////////////////////////////////////////////////////////////////////////
///////////////////////////////////////////////////////////////////////////////
///////////////////////////////////////////////////////////////////////////////
BucleDispositivosTodosMaquina_EventoRecibido_RefrescoDispositivo:NOP   0;


///////////////////////////////////////////////////////////////////////////////
// --- Mirar si esta definido como mesa de Tracking y TL
      SET;
      AN    "DB850_DefinicionMesas".Mesa[#IndiceMaquina].ConfigMesa.MesaPaso;
      AN    "DB850_DefinicionMesas".Mesa[#IndiceMaquina].ConfigMesa.MesaCruce;
      AN    "DB850_DefinicionMesas".Mesa[#IndiceMaquina].ConfigMesa.MesaMultiplesDestinos;
      AN    "DB850_DefinicionMesas".Mesa[#IndiceMaquina].ConfigMesa.MesaTL;
      JC    ContinuarBucleDispositivosTodosMaquina_EventoRecibido_RefrescoDispositivo;


///////////////////////////////////////////////////////////////////////////////
/// Mirar Si hay maquina
      SET;
      AN    "DB850_DefinicionMesas".Mesa[#IndiceMaquina].ConfigMesa.MaquinaEnMesa;  // Maquina ?
      JC    ContinuarBucleDispositivosTodosMaquina_EventoRecibido_RefrescoDispositivo;


///////////////////////////////////////////////////////////////////////////////
/// --- Mirar Si pertenece al JDT
      SET;
      X     "DB850_DefinicionMesas".Mesa[#IndiceMaquina].ConfigMesa.MesaDeJDT02;  // JDT01 ?
      XN    #JDT02_Activo;
      =     #DispositivoDeJDT02;

      SET;
      AN    #DispositivoDeJDT02;
      JC    ContinuarBucleDispositivosTodosMaquina_EventoRecibido_RefrescoDispositivo;


///////////////////////////////////////////////////////////////////////////////
// --- Activar Refresco del Dispositivo
      L     250;  // 250 - Recibido Evento de Refresco de Datos del Dispositivo
      T     "DB832_Maquinas".Maquinas[#IndiceMaquina].EstadoRecepcionEvento;


///////////////////////////////////////////////////////////////////////////////
ContinuarBucleDispositivosTodosMaquina_EventoRecibido_RefrescoDispositivo:NOP   0;
      L     #IndiceMaquina;  // Incremento al siguiente Maquina
      L     1;
      +I;
      T     #IndiceMaquina;

      L     #IndiceMaquina;
      L     "CTE_MaxMesas";
      >I;  // Finalizar
      JC    Final_EventoRecibido_RefrescoDispositivo;


///////////////////////////////////////////////////////////////////////////////
// --- Ir hacia el siguiente Maquina
      JU    BucleDispositivosTodosMaquina_EventoRecibido_RefrescoDispositivo;



NETWORK
TITLE = ---- Accion del Evento --> Peticion de Refresco del Dispositivo Baliza
///////////////////////////////////////////////////////////////////////////////
///////////////////////////////////////////////////////////////////////////////
///////////////////////////////////////////////////////////////////////////////
// Dispositivos tipo Baliza uno determinado o todos
DispositivoBaliza_EventoRecibido_RefrescoDispositivo:NOP   0;
      SET;
      L     #AtributosDeDispositivos.Numero;  // Mirar si hay numero de maquina
      L     0;  // Son todos las Balizas
      ==I;
      JC    DispositivosTodosBaliza_EventoRecibido_RefrescoDispositivo;


///////////////////////////////////////////////////////////////////////////////
// --- Es Una Maquina Determinada
      JU    DispositivosUnaBaliza_EventoRecibido_RefrescoDispositivo;



NETWORK
TITLE = ---- ---- De una Baliza
///////////////////////////////////////////////////////////////////////////////
///////////////////////////////////////////////////////////////////////////////
///////////////////////////////////////////////////////////////////////////////
// --- Una Baliza determinada
DispositivosUnaBaliza_EventoRecibido_RefrescoDispositivo:NOP   0;

      L     #AtributosDeDispositivos.Numero;  // Ver que Baliza es
      L     "CTE_OffsetMesa";
      -I;
      T     #VarTempDispositivos.Numero;

      L     #VarTempDispositivos.Numero;  // Comprobar el numero de Baliza
      L     1;  // No menor de 1
      <I;  // No es correcto
      JC    Final_EventoRecibido_RefrescoDispositivo;
      L     #VarTempDispositivos.Numero;
      L     "CTE_MaxDispositivosBaliza";  // No meyor que el parametro
      >I;  // No es correcto
      JC    Final_EventoRecibido_RefrescoDispositivo;


///////////////////////////////////////////////////////////////////////////////
// --- Activar Refresco del Dispositivo
///////////////////////////////////////////////////////////////////////////////
// Activar Refresco del Dispositivo
      SET;
      S     "DB839_DispositivosVarios".DispoBaliza[#VarTempDispositivos.Numero].RefrescoDatos;


///////////////////////////////////////////////////////////////////////////////
// --- Finalizar
      JU    Final_EventoRecibido_RefrescoDispositivo;



NETWORK
TITLE = ---- ---- De Todas las Balizas
////////////////////////////////////////////////////////////////////////////
////////////////////////////////////////////////////////////////////////////
////////////////////////////////////////////////////////////////////////////
// --- Peticion de Todos los dispositivos BALIZA
DispositivosTodosBaliza_EventoRecibido_RefrescoDispositivo:NOP   0;
      L     1;
      T     #IndiceDispositivosVarios;


////////////////////////////////////////////////////////////////////////////
////////////////////////////////////////////////////////////////////////////
////////////////////////////////////////////////////////////////////////////
BucleBaliza_EventoRecibido_RefrescoDispositivo:NOP   0;


///////////////////////////////////////////////////////////////////////////////
// Activar Refresco del Dispositivo
      SET;
      S     "DB839_DispositivosVarios".DispoBaliza[#IndiceDispositivosVarios].RefrescoDatos;

////////////////////////////////////////////////////////////////////////////
      L     #IndiceDispositivosVarios;  // Siguiente Dispositivo
      L     1;
      +I;
      T     #IndiceDispositivosVarios;

      L     #IndiceDispositivosVarios;
      L     "CTE_MaxDispositivosBaliza";
      >I;  // Ha superado el maximo ??
      JC    FinBucleBaliza_EventoRecibido_RefrescoDispositivo;

      JU    BucleBaliza_EventoRecibido_RefrescoDispositivo;  // Continuar en el Bucle


////////////////////////////////////////////////////////////////////////////
////////////////////////////////////////////////////////////////////////////
////////////////////////////////////////////////////////////////////////////
FinBucleBaliza_EventoRecibido_RefrescoDispositivo:NOP   0;
      JU    Final_EventoRecibido_RefrescoDispositivo;


NETWORK
TITLE = ---- Accion del Evento --> Peticion de Refresco del Dispositivo Llave
///////////////////////////////////////////////////////////////////////////////
///////////////////////////////////////////////////////////////////////////////
///////////////////////////////////////////////////////////////////////////////
// Dispositivos tipo Llave uno determinado o todos
DispositivoLlave_EventoRecibido_RefrescoDispositivo:NOP   0;
      SET;
      L     #AtributosDeDispositivos.Numero;  // Mirar si hay numero de maquina
      L     0;  // Son todos las Llaves
      ==I;
      JC    DispositivosTodosLlave_EventoRecibido_RefrescoDispositivo;


///////////////////////////////////////////////////////////////////////////////
// --- Es Una Maquina Determinada
      JU    DispositivosUnaLlave_EventoRecibido_RefrescoDispositivo;



NETWORK
TITLE = ---- ---- De una Llave
///////////////////////////////////////////////////////////////////////////////
///////////////////////////////////////////////////////////////////////////////
///////////////////////////////////////////////////////////////////////////////
// --- Una Llave determinada
DispositivosUnaLlave_EventoRecibido_RefrescoDispositivo:NOP   0;

      L     #AtributosDeDispositivos.Numero;  // Ver que Llave es
      L     "CTE_OffsetMesa";
      -I;
      T     #VarTempDispositivos.Numero;

      L     #VarTempDispositivos.Numero;  // Comprobar el numero de Llave
      L     1;  // No menor de 1
      <I;  // No es correcto
      JC    Final_EventoRecibido_RefrescoDispositivo;
      L     #VarTempDispositivos.Numero;
      L     "CTE_MaxDispositivosLlave";  // No meyor que el parametro
      >I;  // No es correcto
      JC    Final_EventoRecibido_RefrescoDispositivo;


///////////////////////////////////////////////////////////////////////////////
// --- Activar Refresco del Dispositivo
///////////////////////////////////////////////////////////////////////////////
// Activar Refresco del Dispositivo
      SET;
      S     "DB839_DispositivosVarios".DispoLlave[#VarTempDispositivos.Numero].RefrescoDatos;


///////////////////////////////////////////////////////////////////////////////
// --- Finalizar
      JU    Final_EventoRecibido_RefrescoDispositivo;



NETWORK
TITLE = ---- ---- De Todas las Llaves
////////////////////////////////////////////////////////////////////////////
////////////////////////////////////////////////////////////////////////////
////////////////////////////////////////////////////////////////////////////
// --- Peticion de Todos los dispositivos LLAVE
DispositivosTodosLlave_EventoRecibido_RefrescoDispositivo:NOP   0;
      L     1;
      T     #IndiceDispositivosVarios;


////////////////////////////////////////////////////////////////////////////
////////////////////////////////////////////////////////////////////////////
////////////////////////////////////////////////////////////////////////////
BucleLlave_EventoRecibido_RefrescoDispositivo:NOP   0;


///////////////////////////////////////////////////////////////////////////////
// Activar Refresco del Dispositivo
      SET;
      S     "DB839_DispositivosVarios".DispoLlave[#IndiceDispositivosVarios].RefrescoDatos;
////////////////////////////////////////////////////////////////////////////
      L     #IndiceDispositivosVarios;  // Siguiente Dispositivo
      L     1;
      +I;
      T     #IndiceDispositivosVarios;

      L     #IndiceDispositivosVarios;
      L     "CTE_MaxDispositivosLlave";
      >I;  // Ha superado el maximo ??
      JC    FinBuclellave_EventoRecibido_RefrescoDispositivo;

      JU    BucleLlave_EventoRecibido_RefrescoDispositivo;  // Continuar en el Bucle


////////////////////////////////////////////////////////////////////////////
////////////////////////////////////////////////////////////////////////////
////////////////////////////////////////////////////////////////////////////
FinBuclellave_EventoRecibido_RefrescoDispositivo:NOP   0;
      JU    Final_EventoRecibido_RefrescoDispositivo;


NETWORK
TITLE = ---- Accion del Evento --> Peticion de Refresco del Dispositivo Seta
///////////////////////////////////////////////////////////////////////////////
///////////////////////////////////////////////////////////////////////////////
///////////////////////////////////////////////////////////////////////////////
// Dispositivos tipo Seta uno determinado o todos
DispositivoSeta_EventoRecibido_RefrescoDispositivo:NOP   0;
      SET;
      L     #AtributosDeDispositivos.Numero;  // Mirar si hay numero de maquina
      L     0;  // Son todos las Setas
      ==I;
      JC    DispositivosTodosSeta_EventoRecibido_RefrescoDispositivo;


///////////////////////////////////////////////////////////////////////////////
// --- Es Una Maquina Determinada
      JU    DispositivosUnaSeta_EventoRecibido_RefrescoDispositivo;



NETWORK
TITLE = ---- ---- De una Seta
///////////////////////////////////////////////////////////////////////////////
///////////////////////////////////////////////////////////////////////////////
///////////////////////////////////////////////////////////////////////////////
// --- Una Seta determinada
DispositivosUnaSeta_EventoRecibido_RefrescoDispositivo:NOP   0;

      L     #AtributosDeDispositivos.Numero;  // Ver que Seta es
      L     "CTE_OffsetMesa";
      -I;
      T     #VarTempDispositivos.Numero;

      L     #VarTempDispositivos.Numero;  // Comprobar el numero de Seta
      L     1;  // No menor de 1
      <I;  // No es correcto
      JC    Final_EventoRecibido_RefrescoDispositivo;
      L     #VarTempDispositivos.Numero;
      L     "CTE_MaxDispositivosSeta";  // No meyor que el parametro
      >I;  // No es correcto
      JC    Final_EventoRecibido_RefrescoDispositivo;


///////////////////////////////////////////////////////////////////////////////
// --- Activar Refresco del Dispositivo
///////////////////////////////////////////////////////////////////////////////
// Activar Refresco del Dispositivo
      SET;
      S     "DB839_DispositivosVarios".DispoSeta[#VarTempDispositivos.Numero].RefrescoDatos;


///////////////////////////////////////////////////////////////////////////////
// --- Finalizar
      JU    Final_EventoRecibido_RefrescoDispositivo;



NETWORK
TITLE = ---- ---- De Todas las Setas
////////////////////////////////////////////////////////////////////////////
////////////////////////////////////////////////////////////////////////////
////////////////////////////////////////////////////////////////////////////
// --- Peticion de Todos los dispositivos SETA
DispositivosTodosSeta_EventoRecibido_RefrescoDispositivo:NOP   0;
      L     1;
      T     #IndiceDispositivosVarios;


////////////////////////////////////////////////////////////////////////////
////////////////////////////////////////////////////////////////////////////
////////////////////////////////////////////////////////////////////////////
BucleSeta_EventoRecibido_RefrescoDispositivo:NOP   0;


///////////////////////////////////////////////////////////////////////////////
// Activar Refresco del Dispositivo
      SET;
      S     "DB839_DispositivosVarios".DispoSeta[#IndiceDispositivosVarios].RefrescoDatos;
////////////////////////////////////////////////////////////////////////////
      L     #IndiceDispositivosVarios;  // Siguiente Dispositivo
      L     1;
      +I;
      T     #IndiceDispositivosVarios;

      L     #IndiceDispositivosVarios;
      L     "CTE_MaxDispositivosSeta";
      >I;  // Ha superado el maximo ??
      JC    FinBucleSeta_EventoRecibido_RefrescoDispositivo;

      JU    BucleSeta_EventoRecibido_RefrescoDispositivo;  // Continuar en el Bucle


////////////////////////////////////////////////////////////////////////////
////////////////////////////////////////////////////////////////////////////
////////////////////////////////////////////////////////////////////////////
FinBucleSeta_EventoRecibido_RefrescoDispositivo:NOP   0;
      JU    Final_EventoRecibido_RefrescoDispositivo;


NETWORK
TITLE = ---- Accion del Evento --> Peticion de Refresco del Dispositivo Barrera
///////////////////////////////////////////////////////////////////////////////
///////////////////////////////////////////////////////////////////////////////
///////////////////////////////////////////////////////////////////////////////
// Dispositivos tipo Barrera uno determinado o todos
DispositivoBarrera_EventoRecibido_RefrescoDispositivo:NOP   0;
      SET;
      L     #AtributosDeDispositivos.Numero;  // Mirar si hay numero de maquina
      L     0;  // Son todos las Barreras
      ==I;
      JC    DispositivosTodosBarrera_EventoRecibido_RefrescoDispositivo;


///////////////////////////////////////////////////////////////////////////////
// --- Es Una Maquina Determinada
      JU    DispositivosUnaBarrera_EventoRecibido_RefrescoDispositivo;



NETWORK
TITLE = ---- ---- De una Barrera
///////////////////////////////////////////////////////////////////////////////
///////////////////////////////////////////////////////////////////////////////
///////////////////////////////////////////////////////////////////////////////
// --- Una Barrera  determinada
DispositivosUnaBarrera_EventoRecibido_RefrescoDispositivo:NOP   0;

      L     #AtributosDeDispositivos.Numero;  // Ver que Barrera es
      L     "CTE_OffsetMesa";
      -I;
      T     #VarTempDispositivos.Numero;

      L     #VarTempDispositivos.Numero;  // Comprobar el numero de Barrera
      L     1;  // No menor de 1
      <I;  // No es correcto
      JC    Final_EventoRecibido_RefrescoDispositivo;
      L     #VarTempDispositivos.Numero;
      L     "CTE_MaxDispositivosBarrera";  // No meyor que el parametro
      >I;  // No es correcto
      JC    Final_EventoRecibido_RefrescoDispositivo;


///////////////////////////////////////////////////////////////////////////////
// --- Activar Refresco del Dispositivo
///////////////////////////////////////////////////////////////////////////////
// Activar Refresco del Dispositivo
      SET;
      S     "DB839_DispositivosVarios".DispoBarrera[#VarTempDispositivos.Numero].RefrescoDatos;


///////////////////////////////////////////////////////////////////////////////
// --- Finalizar
      JU    Final_EventoRecibido_RefrescoDispositivo;



NETWORK
TITLE = ---- ---- De Todas las Barreras
////////////////////////////////////////////////////////////////////////////
////////////////////////////////////////////////////////////////////////////
////////////////////////////////////////////////////////////////////////////
// --- Peticion de Todos los dispositivos BARRERA
DispositivosTodosBarrera_EventoRecibido_RefrescoDispositivo:NOP   0;
      L     1;
      T     #IndiceDispositivosVarios;


////////////////////////////////////////////////////////////////////////////
////////////////////////////////////////////////////////////////////////////
////////////////////////////////////////////////////////////////////////////
BucleBarrera_EventoRecibido_RefrescoDispositivo:NOP   0;


///////////////////////////////////////////////////////////////////////////////
// Activar Refresco del Dispositivo
      SET;
      S     "DB839_DispositivosVarios".DispoBarrera[#IndiceDispositivosVarios].RefrescoDatos;
////////////////////////////////////////////////////////////////////////////
      L     #IndiceDispositivosVarios;  // Siguiente Dispositivo
      L     1;
      +I;
      T     #IndiceDispositivosVarios;

      L     #IndiceDispositivosVarios;
      L     "CTE_MaxDispositivosBarrera";
      >I;  // Ha superado el maximo ??
      JC    FinBucleBarrera_EventoRecibido_RefrescoDispositivo;

      JU    BucleBarrera_EventoRecibido_RefrescoDispositivo;  // Continuar en el Bucle


////////////////////////////////////////////////////////////////////////////
////////////////////////////////////////////////////////////////////////////
////////////////////////////////////////////////////////////////////////////
FinBucleBarrera_EventoRecibido_RefrescoDispositivo:NOP   0;
      JU    Final_EventoRecibido_RefrescoDispositivo;


NETWORK
TITLE = ---- Accion del Evento --> Peticion de Refresco del Dispositivo Puerta
///////////////////////////////////////////////////////////////////////////////
///////////////////////////////////////////////////////////////////////////////
///////////////////////////////////////////////////////////////////////////////
// Dispositivos tipo Puerta uno determinado o todos
DispositivoPuerta_EventoRecibido_RefrescoDispositivo:NOP   0;
      SET;
      L     #AtributosDeDispositivos.Numero;  // Mirar si hay numero de maquina
      L     0;  // Son todos las Puertas
      ==I;
      JC    DispositivosTodosPuerta_EventoRecibido_RefrescoDispositivo;


///////////////////////////////////////////////////////////////////////////////
// --- Es Una Maquina Determinada
      JU    DispositivosUnaPuerta_EventoRecibido_RefrescoDispositivo;



NETWORK
TITLE = ---- ---- De una Puerta
///////////////////////////////////////////////////////////////////////////////
///////////////////////////////////////////////////////////////////////////////
///////////////////////////////////////////////////////////////////////////////
// --- Uan Puerta determinada
DispositivosUnaPuerta_EventoRecibido_RefrescoDispositivo:NOP   0;

      L     #AtributosDeDispositivos.Numero;  // Ver que Puerta es
      L     "CTE_OffsetMesa";
      -I;
      T     #VarTempDispositivos.Numero;

      L     #VarTempDispositivos.Numero;  // Comprobar el numero de Puerta
      L     1;  // No menor de 1
      <I;  // No es correcto
      JC    Final_EventoRecibido_RefrescoDispositivo;
      L     #VarTempDispositivos.Numero;
      L     "CTE_MaxDispositivosPuerta";  // No meyor que el parametro
      >I;  // No es correcto
      JC    Final_EventoRecibido_RefrescoDispositivo;


///////////////////////////////////////////////////////////////////////////////
// --- Activar Refresco del Dispositivo
///////////////////////////////////////////////////////////////////////////////
// Activar Refresco del Dispositivo
      SET;
      S     "DB839_DispositivosVarios".DispoPuerta[#VarTempDispositivos.Numero].RefrescoDatos;


///////////////////////////////////////////////////////////////////////////////
// --- Finalizar
      JU    Final_EventoRecibido_RefrescoDispositivo;



NETWORK
TITLE = ---- ---- De Todas las Puertas
////////////////////////////////////////////////////////////////////////////
////////////////////////////////////////////////////////////////////////////
////////////////////////////////////////////////////////////////////////////
// --- Peticion de Todos los dispositivos PUERTA
DispositivosTodosPuerta_EventoRecibido_RefrescoDispositivo:NOP   0;
      L     1;
      T     #IndiceDispositivosVarios;


////////////////////////////////////////////////////////////////////////////
////////////////////////////////////////////////////////////////////////////
////////////////////////////////////////////////////////////////////////////
BuclePuerta_EventoRecibido_RefrescoDispositivo:NOP   0;


///////////////////////////////////////////////////////////////////////////////
// Activar Refresco del Dispositivo
      SET;
      S     "DB839_DispositivosVarios".DispoPuerta[#IndiceDispositivosVarios].RefrescoDatos;

////////////////////////////////////////////////////////////////////////////
      L     #IndiceDispositivosVarios;  // Siguiente Dispositivo
      L     1;
      +I;
      T     #IndiceDispositivosVarios;

      L     #IndiceDispositivosVarios;
      L     "CTE_MaxDispositivosPuerta";
      >I;  // Ha superado el maximo ??
      JC    FinBuclePuerta_EventoRecibido_RefrescoDispositivo;

      JU    BuclePuerta_EventoRecibido_RefrescoDispositivo;  // Continuar en el Bucle


////////////////////////////////////////////////////////////////////////////
////////////////////////////////////////////////////////////////////////////
////////////////////////////////////////////////////////////////////////////
FinBuclePuerta_EventoRecibido_RefrescoDispositivo:NOP   0;
      JU    Final_EventoRecibido_RefrescoDispositivo;


NETWORK
TITLE = ---- Accion del Evento --> Peticion de Refresco del Dispositivo Linea de Potencia
///////////////////////////////////////////////////////////////////////////////
///////////////////////////////////////////////////////////////////////////////
///////////////////////////////////////////////////////////////////////////////
// Dispositivos tipo Linea de Potencia uno determinado o todos
DispositivoLineaPotencia_EventoRecibido_RefrescoDispositivo:NOP   0;
      SET;
      L     #AtributosDeDispositivos.Numero;  // Mirar si hay numero de maquina
      L     0;  // Son todos las Lineas de Potencia
      ==I;
      JC    DispositivosTodosLineaPotencia_EventoRecibido_RefrescoDispositivo;


///////////////////////////////////////////////////////////////////////////////
// --- Es Una Maquina Determinada
      JU    DispositivosUnaLineaPotencia_EventoRecibido_RefrescoDispositivo;



NETWORK
TITLE = ---- ---- De una Linea de Potencia
///////////////////////////////////////////////////////////////////////////////
///////////////////////////////////////////////////////////////////////////////
///////////////////////////////////////////////////////////////////////////////
// --- Maquina  determinada
DispositivosUnaLineaPotencia_EventoRecibido_RefrescoDispositivo:NOP   0;

      L     #AtributosDeDispositivos.Numero;  // Ver que Linea de Potencia es
      L     "CTE_OffsetMesa";
      -I;
      T     #VarTempDispositivos.Numero;

      L     #VarTempDispositivos.Numero;  // Comprobar el numero de Linea de Potencia
      L     1;  // No menor de 1
      <I;  // No es correcto
      JC    Final_EventoRecibido_RefrescoDispositivo;
      L     #VarTempDispositivos.Numero;
      L     "CTE_MaxDispositivosLineaPotencia";  // No meyor que el parametro
      >I;  // No es correcto
      JC    Final_EventoRecibido_RefrescoDispositivo;


///////////////////////////////////////////////////////////////////////////////
// --- Activar Refresco del Dispositivo
///////////////////////////////////////////////////////////////////////////////
// Activar Refresco del Dispositivo
      SET;
      S     "DB839_DispositivosVarios".DispoLineaPotencia[#VarTempDispositivos.Numero].RefrescoDatos;


///////////////////////////////////////////////////////////////////////////////
// --- Finalizar
      JU    Final_EventoRecibido_RefrescoDispositivo;



NETWORK
TITLE = ---- ---- De Todas Las Lineas de Potencia
////////////////////////////////////////////////////////////////////////////
////////////////////////////////////////////////////////////////////////////
////////////////////////////////////////////////////////////////////////////
// --- Peticion de Todos los dispositivos LINEA DE POTENCIA
DispositivosTodosLineaPotencia_EventoRecibido_RefrescoDispositivo:NOP   0;
      L     1;
      T     #IndiceDispositivosVarios;


////////////////////////////////////////////////////////////////////////////
////////////////////////////////////////////////////////////////////////////
////////////////////////////////////////////////////////////////////////////
BucleLineaPotencia_EventoRecibido_RefrescoDispositivo:NOP   0;


///////////////////////////////////////////////////////////////////////////////
// Activar Refresco del Dispositivo
      SET;
      S     "DB839_DispositivosVarios".DispoLineaPotencia[#IndiceDispositivosVarios].RefrescoDatos;

////////////////////////////////////////////////////////////////////////////
      L     #IndiceDispositivosVarios;  // Siguiente Dispositivo
      L     1;
      +I;
      T     #IndiceDispositivosVarios;

      L     #IndiceDispositivosVarios;
      L     "CTE_MaxDispositivosLineaPotencia";
      >I;  // Ha superado el maximo ??
      JC    FinBucleLineaPotencia_EventoRecibido_RefrescoDispositivo;

      JU    BucleLineaPotencia_EventoRecibido_RefrescoDispositivo;  // Continuar en el Bucle


////////////////////////////////////////////////////////////////////////////
////////////////////////////////////////////////////////////////////////////
////////////////////////////////////////////////////////////////////////////
FinBucleLineaPotencia_EventoRecibido_RefrescoDispositivo:NOP   0;
      JU    Final_EventoRecibido_RefrescoDispositivo;


NETWORK
TITLE = ---- Accion del Evento --> Peticion de Refresco de Todos Los Dispositivos
///////////////////////////////////////////////////////////////////////////////
///////////////////////////////////////////////////////////////////////////////
///////////////////////////////////////////////////////////////////////////////
// --- Todos los dispositivos
DispositivosTodos_EventoRecibido_RefrescoDispositivo:NOP   0;



NETWORK
TITLE = ---- ---- CCPIF y CBOX
///////////////////////////////////////////////////////////////////////////////
///////////////////////////////////////////////////////////////////////////////
///////////////////////////////////////////////////////////////////////////////
// --- Recorrer CCPIF y Todos los CBOX
      L     0;
      T     #IndiceCBOX;


///////////////////////////////////////////////////////////////////////////////
///////////////////////////////////////////////////////////////////////////////
///////////////////////////////////////////////////////////////////////////////
BucleArmarios_DispositivosTodos_EventoRecibido_RefrescoDispositivo:NOP   0;


///////////////////////////////////////////////////////////////////////////////
/// --- Inicio si pertenece al JDT
      SET;
      X     "DB855_DefinicionDispositivos".Dispositivos[#IndiceCBOX].EventosDelJdT02;
      XN    #JDT02_Activo;
      =     #DispositivoDeJDT02;

      SET;
      AN    #DispositivoDeJDT02;
      JC    ContinuarBucleArmarios_DispositivosTodos_EventoRecibido_RefrescoDispositivo;


///////////////////////////////////////////////////////////////////////////////
// --- Activar Refresco del Dispositivo
      L     250;  // 250 - Recibido Evento de Refresco de Datos del Dispositivo
      T     "DB830_Dispositivos".Dispositivos[#IndiceCBOX].EstadoRecepcionEvento;


///////////////////////////////////////////////////////////////////////////////
ContinuarBucleArmarios_DispositivosTodos_EventoRecibido_RefrescoDispositivo:NOP   0;
      L     #IndiceCBOX;  // Incremento al siguiente CBOX
      L     1;
      +I;
      T     #IndiceCBOX;

      L     #IndiceCBOX;
      L     "CTE_MaxDispositivos";
      >I;  // Finalizar
      JC    FinBucleArmarios_DispositivosTodos_EventoRecibido_RefrescoDispositivos;

///////////////////////////////////////////////////////////////////////////////
// --- Ir hacia el siguiente CBOX
      JU    BucleArmarios_DispositivosTodos_EventoRecibido_RefrescoDispositivo;


///////////////////////////////////////////////////////////////////////////////
///////////////////////////////////////////////////////////////////////////////
///////////////////////////////////////////////////////////////////////////////
FinBucleArmarios_DispositivosTodos_EventoRecibido_RefrescoDispositivos:NOP   0;



NETWORK
TITLE = ---- ---- Mesas
///////////////////////////////////////////////////////////////////////////////
///////////////////////////////////////////////////////////////////////////////
// Recorrer Todas las Mesas
      L     1;
      T     #IndiceMesa;

///////////////////////////////////////////////////////////////////////////////
///////////////////////////////////////////////////////////////////////////////
///////////////////////////////////////////////////////////////////////////////
BucleMesas_DispositivosTodos_EventoRecibido_RefrescoDispositivo:NOP   0;


///////////////////////////////////////////////////////////////////////////////
// --- Mirar si esta definido como mesa de Tracking y TL
      SET;
      AN    "DB850_DefinicionMesas".Mesa[#IndiceMesa].ConfigMesa.MesaPaso;
      AN    "DB850_DefinicionMesas".Mesa[#IndiceMesa].ConfigMesa.MesaCruce;
      AN    "DB850_DefinicionMesas".Mesa[#IndiceMesa].ConfigMesa.MesaMultiplesDestinos;
      AN    "DB850_DefinicionMesas".Mesa[#IndiceMesa].ConfigMesa.MesaTL;
      JC    ContinuarBucleMesas_DispositivosTodos_EventoRecibido_RefrescoDispositivo;


///////////////////////////////////////////////////////////////////////////////
// --- Mirar Si pertenece al JDT
      SET;
      X     "DB850_DefinicionMesas".Mesa[#IndiceMesa].ConfigMesa.MesaDeJDT02;  // JDT01 ?
      XN    #JDT02_Activo;
      =     #DispositivoDeJDT02;

      SET;
      AN    #DispositivoDeJDT02;
      JC    ContinuarBucleMesas_DispositivosTodos_EventoRecibido_RefrescoDispositivo;


///////////////////////////////////////////////////////////////////////////////
// --- Activar Refresco del Dispositivo
      L     250;  // 250 - Recibido Evento de Refresco de Datos del Dispositivo
      T     "DB831_Mesas".Mesas[#IndiceMesa].EstadoRecepcionEvento;


///////////////////////////////////////////////////////////////////////////////
ContinuarBucleMesas_DispositivosTodos_EventoRecibido_RefrescoDispositivo:NOP   0;

      L     #IndiceMesa;  // Incremento al siguiente Mesa
      L     1;
      +I;
      T     #IndiceMesa;

      L     #IndiceMesa;
      L     "CTE_MaxMesas";
      >I;  // Finalizar
      JC    FinBucleMesas_DispositivosTodos_EventoRecibido_RefrescoDispositivo;


///////////////////////////////////////////////////////////////////////////////
// --- Ir hacia el siguiente Mesa
      JU    BucleMesas_DispositivosTodos_EventoRecibido_RefrescoDispositivo;


///////////////////////////////////////////////////////////////////////////////
///////////////////////////////////////////////////////////////////////////////
///////////////////////////////////////////////////////////////////////////////
FinBucleMesas_DispositivosTodos_EventoRecibido_RefrescoDispositivo:NOP   0;



NETWORK
TITLE = ---- ---- Maquinas
///////////////////////////////////////////////////////////////////////////////
///////////////////////////////////////////////////////////////////////////////
///////////////////////////////////////////////////////////////////////////////
// Recorrer todas las Maquinas
      L     1;
      T     #IndiceMaquina;


///////////////////////////////////////////////////////////////////////////////
///////////////////////////////////////////////////////////////////////////////
///////////////////////////////////////////////////////////////////////////////
BucleMaquinas_DispositivosTodos_EventoRecibido_RefrescoDispositivo:NOP   0;


///////////////////////////////////////////////////////////////////////////////
// --- Mirar si esta definido como mesa de Tracking y TL
      SET;
      AN    "DB850_DefinicionMesas".Mesa[#IndiceMaquina].ConfigMesa.MesaPaso;
      AN    "DB850_DefinicionMesas".Mesa[#IndiceMaquina].ConfigMesa.MesaCruce;
      AN    "DB850_DefinicionMesas".Mesa[#IndiceMaquina].ConfigMesa.MesaMultiplesDestinos;
      AN    "DB850_DefinicionMesas".Mesa[#IndiceMaquina].ConfigMesa.MesaTL;
      JC    ContinuarBucleMaquinas_DispositivosTodos_EventoRecibido_RefrescoDispositivo;


///////////////////////////////////////////////////////////////////////////////
/// --- Mirar Si hay maquina
      SET;
      AN    "DB850_DefinicionMesas".Mesa[#IndiceMaquina].ConfigMesa.MaquinaEnMesa;  // Maquina ?
      JC    ContinuarBucleMaquinas_DispositivosTodos_EventoRecibido_RefrescoDispositivo;


///////////////////////////////////////////////////////////////////////////////
/// --- Mirar Si pertenece al JDT
      SET;
      X     "DB850_DefinicionMesas".Mesa[#IndiceMaquina].ConfigMesa.MesaDeJDT02;  // JDT01 ?
      XN    #JDT02_Activo;
      =     #MesaDeJDT02;

      SET;
      AN    #MesaDeJDT02;
      JC    ContinuarBucleMaquinas_DispositivosTodos_EventoRecibido_RefrescoDispositivo;


///////////////////////////////////////////////////////////////////////////////
// Activar Refresco del Dispositivo
      L     250;  // 250 - Recibido Evento de Refresco de Datos del Dispositivo
      T     "DB832_Maquinas".Maquinas[#IndiceMaquina].EstadoRecepcionEvento;


///////////////////////////////////////////////////////////////////////////////
ContinuarBucleMaquinas_DispositivosTodos_EventoRecibido_RefrescoDispositivo:NOP   0;
      L     #IndiceMaquina;  // Incremento al siguiente Maquina
      L     1;
      +I;
      T     #IndiceMaquina;

      L     #IndiceMaquina;
      L     "CTE_MaxMesas";
      >I;  // Finalizar
      JC    FinBucleMaquinas_DispositivosTodos_EventoRecibido_RefrescoDispositivo;


///////////////////////////////////////////////////////////////////////////////
// --- Ir hacia el siguiente Maquina
      JU    BucleMaquinas_DispositivosTodos_EventoRecibido_RefrescoDispositivo;


///////////////////////////////////////////////////////////////////////////////
///////////////////////////////////////////////////////////////////////////////
///////////////////////////////////////////////////////////////////////////////
FinBucleMaquinas_DispositivosTodos_EventoRecibido_RefrescoDispositivo:NOP   0;



NETWORK
TITLE = ---- ---- Balizas
////////////////////////////////////////////////////////////////////////////
////////////////////////////////////////////////////////////////////////////
////////////////////////////////////////////////////////////////////////////
// --- Peticion de Todos los dispositivos BALIZA

      L     1;
      T     #IndiceDispositivosVarios;


////////////////////////////////////////////////////////////////////////////
////////////////////////////////////////////////////////////////////////////
////////////////////////////////////////////////////////////////////////////
BucleBaliza_DispositivosTodos_EventoRecibido_RefrescoDispositivo:NOP   0;


///////////////////////////////////////////////////////////////////////////////
// Activar Refresco del Dispositivo
      SET;
      S     "DB839_DispositivosVarios".DispoBaliza[#IndiceDispositivosVarios].RefrescoDatos;
////////////////////////////////////////////////////////////////////////////
      L     #IndiceDispositivosVarios;  // Siguiente Dispositivo
      L     1;
      +I;
      T     #IndiceDispositivosVarios;

      L     #IndiceDispositivosVarios;
      L     "CTE_MaxDispositivosBaliza";
      >I;  // Ha superado el maximo ??
      JC    FinBucleBaliza_DispositivosTodos_EventoRecibido_RefrescoDispositivo;

      JU    BucleBaliza_DispositivosTodos_EventoRecibido_RefrescoDispositivo;  // Continuar en el Bucle


////////////////////////////////////////////////////////////////////////////
////////////////////////////////////////////////////////////////////////////
////////////////////////////////////////////////////////////////////////////
FinBucleBaliza_DispositivosTodos_EventoRecibido_RefrescoDispositivo:NOP   0;



NETWORK
TITLE = ---- ---- Llaves
////////////////////////////////////////////////////////////////////////////
////////////////////////////////////////////////////////////////////////////
////////////////////////////////////////////////////////////////////////////
// --- Peticion de Todos los dispositivos LLAVE

      L     1;
      T     #IndiceDispositivosVarios;


////////////////////////////////////////////////////////////////////////////
////////////////////////////////////////////////////////////////////////////
////////////////////////////////////////////////////////////////////////////
BucleLlave_DispositivosTodos_EventoRecibido_RefrescoDispositivo:NOP   0;


///////////////////////////////////////////////////////////////////////////////
// Activar Refresco del Dispositivo
      SET;
      S     "DB839_DispositivosVarios".DispoLlave[#IndiceDispositivosVarios].RefrescoDatos;
////////////////////////////////////////////////////////////////////////////
      L     #IndiceDispositivosVarios;  // Siguiente Dispositivo
      L     1;
      +I;
      T     #IndiceDispositivosVarios;

      L     #IndiceDispositivosVarios;
      L     "CTE_MaxDispositivosLlave";
      >I;  // Ha superado el maximo ??
      JC    FinBuclellave_DispositivosTodos_EventoRecibido_RefrescoDispositivo;

      JU    BucleLlave_DispositivosTodos_EventoRecibido_RefrescoDispositivo;  // Continuar en el Bucle


////////////////////////////////////////////////////////////////////////////
////////////////////////////////////////////////////////////////////////////
////////////////////////////////////////////////////////////////////////////
FinBuclellave_DispositivosTodos_EventoRecibido_RefrescoDispositivo:NOP   0;



NETWORK
TITLE = ---- ---- Setas
////////////////////////////////////////////////////////////////////////////
////////////////////////////////////////////////////////////////////////////
////////////////////////////////////////////////////////////////////////////
// --- Peticion de Todos los dispositivos SETA

      L     1;
      T     #IndiceDispositivosVarios;


////////////////////////////////////////////////////////////////////////////
////////////////////////////////////////////////////////////////////////////
////////////////////////////////////////////////////////////////////////////
BucleSeta_DispositivosTodos_EventoRecibido_RefrescoDispositivo:NOP   0;


///////////////////////////////////////////////////////////////////////////////
// Activar Refresco del Dispositivo
      SET;
      S     "DB839_DispositivosVarios".DispoSeta[#IndiceDispositivosVarios].RefrescoDatos;
////////////////////////////////////////////////////////////////////////////
      L     #IndiceDispositivosVarios;  // Siguiente Dispositivo
      L     1;
      +I;
      T     #IndiceDispositivosVarios;

      L     #IndiceDispositivosVarios;
      L     "CTE_MaxDispositivosSeta";
      >I;  // Ha superado el maximo ??
      JC    FinBucleSeta_DispositivosTodos_EventoRecibido_RefrescoDispositivo;

      JU    BucleSeta_DispositivosTodos_EventoRecibido_RefrescoDispositivo;  // Continuar en el Bucle


////////////////////////////////////////////////////////////////////////////
////////////////////////////////////////////////////////////////////////////
////////////////////////////////////////////////////////////////////////////
FinBucleSeta_DispositivosTodos_EventoRecibido_RefrescoDispositivo:NOP   0;



NETWORK
TITLE = ---- ---- Barreras
////////////////////////////////////////////////////////////////////////////
////////////////////////////////////////////////////////////////////////////
////////////////////////////////////////////////////////////////////////////
// --- Peticion de Todos los dispositivos BARRERA

      L     1;
      T     #IndiceDispositivosVarios;


////////////////////////////////////////////////////////////////////////////
////////////////////////////////////////////////////////////////////////////
////////////////////////////////////////////////////////////////////////////
BucleBarrera_DispositivosTodos_EventoRecibido_RefrescoDispositivo:NOP   0;


///////////////////////////////////////////////////////////////////////////////
// Activar Refresco del Dispositivo
      SET;
      S     "DB839_DispositivosVarios".DispoBarrera[#IndiceDispositivosVarios].RefrescoDatos;
////////////////////////////////////////////////////////////////////////////
      L     #IndiceDispositivosVarios;  // Siguiente Dispositivo
      L     1;
      +I;
      T     #IndiceDispositivosVarios;

      L     #IndiceDispositivosVarios;
      L     "CTE_MaxDispositivosBarrera";
      >I;  // Ha superado el maximo ??
      JC    FinBucleBarrera_DispositivosTodos_EventoRecibido_RefrescoDispositivo;

      JU    BucleBarrera_DispositivosTodos_EventoRecibido_RefrescoDispositivo;  // Continuar en el Bucle


////////////////////////////////////////////////////////////////////////////
////////////////////////////////////////////////////////////////////////////
////////////////////////////////////////////////////////////////////////////
FinBucleBarrera_DispositivosTodos_EventoRecibido_RefrescoDispositivo:NOP   0;



NETWORK
TITLE = ---- ---- Puertas
////////////////////////////////////////////////////////////////////////////
////////////////////////////////////////////////////////////////////////////
////////////////////////////////////////////////////////////////////////////
// --- Peticion de Todos los dispositivos PUERTA

      L     1;
      T     #IndiceDispositivosVarios;


////////////////////////////////////////////////////////////////////////////
////////////////////////////////////////////////////////////////////////////
////////////////////////////////////////////////////////////////////////////
BuclePuerta_DispositivosTodos_EventoRecibido_RefrescoDispositivo:NOP   0;


///////////////////////////////////////////////////////////////////////////////
// Activar Refresco del Dispositivo
      SET;
      S     "DB839_DispositivosVarios".DispoPuerta[#IndiceDispositivosVarios].RefrescoDatos;
////////////////////////////////////////////////////////////////////////////
      L     #IndiceDispositivosVarios;  // Siguiente Dispositivo
      L     1;
      +I;
      T     #IndiceDispositivosVarios;

      L     #IndiceDispositivosVarios;
      L     "CTE_MaxDispositivosPuerta";
      >I;  // Ha superado el maximo ??
      JC    FinBuclePuerta_DispositivosTodos_EventoRecibido_RefrescoDispositivo;

      JU    BuclePuerta_DispositivosTodos_EventoRecibido_RefrescoDispositivo;  // Continuar en el Bucle


////////////////////////////////////////////////////////////////////////////
////////////////////////////////////////////////////////////////////////////
////////////////////////////////////////////////////////////////////////////
FinBuclePuerta_DispositivosTodos_EventoRecibido_RefrescoDispositivo:NOP   0;



NETWORK
TITLE = ---- ---- Linea de Potencia
////////////////////////////////////////////////////////////////////////////
////////////////////////////////////////////////////////////////////////////
////////////////////////////////////////////////////////////////////////////
// --- Peticion de Todos los dispositivos LINEA DE POTENCIA

      L     1;
      T     #IndiceDispositivosVarios;


////////////////////////////////////////////////////////////////////////////
////////////////////////////////////////////////////////////////////////////
////////////////////////////////////////////////////////////////////////////
BucleLineaPotencia_DispositivosTodos_EventoRecibido_RefrescoDispositivo:NOP   0;


///////////////////////////////////////////////////////////////////////////////
// Activar Refresco del Dispositivo
      SET;
      S     "DB839_DispositivosVarios".DispoLineaPotencia[#IndiceDispositivosVarios].RefrescoDatos;
////////////////////////////////////////////////////////////////////////////
      L     #IndiceDispositivosVarios;  // Siguiente Dispositivo
      L     1;
      +I;
      T     #IndiceDispositivosVarios;

      L     #IndiceDispositivosVarios;
      L     "CTE_MaxDispositivosLineaPotencia";
      >I;  // Ha superado el maximo ??
      JC    FinBucleLineaPotencia_DispositivosTodos_EventoRecibido_RefrescoDispositivo;

      JU    BucleLineaPotencia_DispositivosTodos_EventoRecibido_RefrescoDispositivo;  // Continuar en el Bucle


////////////////////////////////////////////////////////////////////////////
////////////////////////////////////////////////////////////////////////////
////////////////////////////////////////////////////////////////////////////
FinBucleLineaPotencia_DispositivosTodos_EventoRecibido_RefrescoDispositivo:NOP   0;



NETWORK
TITLE = ---- Final
///////////////////////////////////////////////////////////////////////////////
///////////////////////////////////////////////////////////////////////////////
///////////////////////////////////////////////////////////////////////////////
// --- Se acabo el evento
Final_EventoRecibido_RefrescoDispositivo:NOP   0;
      L     #P_Eventos;  // Recupero por donde voy en la lista de eventos
      LAR2;  // Regreso a buscar el siguiente evento
      JU    FinBucle_EventosRecibidos;



NETWORK
TITLE = Evento DID0 - Notificacion de Cambio de Estado de Trabajo de un Dispositivo
// Analisis del evento
// - Inicializa variables de los atributos del Evento
// - Buscar Atributos o Final del Evento
// - Guardar datos del Evento
//   - Si es tipo CCPIF (50)
//   - Si es tipo CBOX (40)
//   - Si es tipo Mesa (60)
//   - Si es tipo Maquina (70)
// Analisis de los atributos de los eventos
// - Mirar que atributo del Evento es ?
// - Distribuir a recoger los datos del Evento
// - Recoger el Atributo Tipo de Dispositivo
// - Recoger el Atributo Numero de Dispositivo
// - Recoger el Atributo Nuevo Estado del Dispositivo
GuardarDatos_EventoRecibido_DIDO:NOP   0;

/////////////////////////////////////////////////////////////////////////
/////////////////////////////////////////////////////////////////////////
/////////////////////////////////////////////////////////////////////////
// --- Guardar Datos del Evento Recibido


/////////////////////////////////////////////////////////////////////////
/////////////////////////////////////////////////////////////////////////
/////////////////////////////////////////////////////////////////////////
/// --- Repartir segun tipo de dispositivo: CCPIF, CBOX, Mesa ...

      SET;  // Es CCPIF
      L     #AtributosDeDispositivos.Tipo;
      L     50;
      ==I;
      JC    DispositivoCCPIF_EventoRecibido_DIDO;

      SET;  // Es CBOX
      L     #AtributosDeDispositivos.Tipo;
      L     40;
      ==I;
      JC    DispositivoCBOX_EventoRecibido_DIDO;

      SET;  // Es Mesa
      L     #AtributosDeDispositivos.Tipo;
      L     60;
      ==I;
      JC    DispositivoMesa_EventoRecibido_DIDO;


/////////////////////////////////////////////////////////////////////////
/////////////////////////////////////////////////////////////////////////
/////////////////////////////////////////////////////////////////////////

      SET;  // Es VTDC
      L     #AtributosDeDispositivos.Tipo;
      L     "CTE_TipoMaquinaVTDC";
      ==I;
      JC    Dispositivo_VTDC_ELEV_EventoRecibido_DIDO;
      SET;  // Es ELEV
      L     #AtributosDeDispositivos.Tipo;
      L     "CTE_TipoMaquinaELEV";
      ==I;
      JC    Dispositivo_VTDC_ELEV_EventoRecibido_DIDO;

// Es Maquina 70 ... 99
      SET;
      A(;
      L     #AtributosDeDispositivos.Tipo;
      L     70;
      >=I;
      );
      A(;
      L     #AtributosDeDispositivos.Tipo;
      L     99;
      <=I;
      );
      JC    DispositivoMaquina_EventoRecibido_DIDO;


/////////////////////////////////////////////////////////////////////////
/////////////////////////////////////////////////////////////////////////
/////////////////////////////////////////////////////////////////////////
// No es ningun Tipo de Dispositivo esperado
      JU    Final_EventoRecibido_DIDO;



NETWORK
TITLE = ---- Accion del Evento --> Notificacion de Cambio de Estado de Trabajo del CCPIF
///////////////////////////////////////////////////////////////////////////////
///////////////////////////////////////////////////////////////////////////////
// --- Tipo CCPIF
DispositivoCCPIF_EventoRecibido_DIDO:NOP   0;
      L     #AtributosDeDispositivos.Numero;  // Comprobacion del numero de CCPIF
      L     "CTE_OffsetCCPIF";
      -I;
      L     1;
      <>I;  // Numero de CCPIF incorrecto
      JC    Final_EventoRecibido_DIDO;




// ????? -------------- ?????
// ????? Por ahora nada ?????
// ????? -------------- ?????




